DATA_BLOCK "08_AL_FILTER"
{ DB_Accessible_From_OPC_UA := 'FALSE' ;
 DB_Accessible_From_Webserver := 'FALSE' ;
 S7_Optimized_Access := 'TRUE' }
VERSION : 0.1
NON_RETAIN
   VAR
      "n0003-mc1-k3201_SN10" : Bool;
      "n0014-pc4-K3001_SN10" : Bool;
   END_VAR


BEGIN

END_DATA_BLOCK

